# EPICS autosave request: trunk/stdApp/Db/countDownTimer_settings.req
# FILE... countDowntTimer_settings.req
$(P)cdt$(N):upDown
$(P)cdt$(N):setTimeHrs
$(P)cdt$(N):setTimeMin
$(P)cdt$(N):setTimeSec
$(P)cdt$(N):trigger.OUT
